// TIA Portal V18 export
FUNCTION "1SecEdgePulse" : Void   // FC59999, LAD
{ S7_Optimized_Access := 'TRUE' }
VERSION : 0.1
// stored: AutoNumber false, IsIECCheckEnabled false, SetENOAutomatically false, UDAEnableTagReadback false
BEGIN

REGION Network 1: Одноразовий імпуьс 1сек
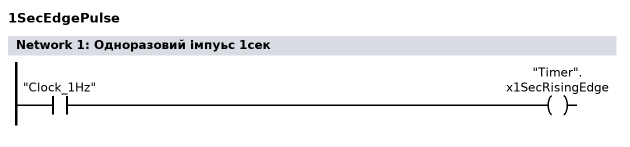
   RUNG wire#powerrail
      Contact( "Clock_1Hz" )
      Coil( "Timer".x1SecRisingEdge )
   END_RUNG
   // the same network as SCL:
   "Timer".x1SecRisingEdge := "Clock_1Hz";
END_REGION

REGION Network 2 (SCL)
   "Timer".x1SecRisingEdge := ("Clock_1Hz" AND NOT "Timer".x1SecPrevClock) AND NOT "Timer".x1SecFired;
   "Timer".x1SecPrevClock := "Clock_1Hz";
   IF "Timer".x1SecRisingEdge THEN
       "Timer".x1SecFired := TRUE;
   END_IF;
END_REGION
END_FUNCTION
